// TIA Portal V17 export
// export: Created 2021-12-03T08:13:09.0752717Z, ExportSetting WithDefaults, DisplayName Totally Integrated Automation Portal, DisplayVersion V17, DisplayName TIA Portal Openness, DisplayVersion V17, DisplayName TIA Portal Version Control Interface, DisplayVersion V17, DisplayName STEP 7 Professional, DisplayVersion V17, DisplayName STEP 7 Safety, DisplayVersion V17, DisplayName WinCC Advanced, DisplayVersion V17
DATA_BLOCK "DBI_Flt_ConvCyclTime"   // DB43
VERSION : 0.1
// stored: AutoNumber false, InstanceOfName FB_FitMem, InstanceOfType FB
"FB_FitMem"
   // VAR_INPUT
   //    I_Ack : Bool;
   //    I_Fit : Bool;
   // END_VAR
   // VAR_OUTPUT
   //    O_Fit : Bool;
   //    O_AskRq : Bool;
   // END_VAR
   // VAR RETAIN
   //    S_AxVar_Pedg_Ack : Bool;
   //    S_AxVar_RSFF_Flt : Bool;
   //    S_Flt : Bool;
   // END_VAR
BEGIN
END_DATA_BLOCK
